% RSLogix 500 project ANALOG PID HEATER CONTROL.RSS, saved by version 8.30.00.16 %
PROJECT "HEATER"    % processor: Bul.1763 MicroLogix 1100 Series B %

PROGRAM FILES
  LAD 2   6 rungs

DATA FILES
  O0 OUTPUT  8 elements
  I1 INPUT  15 elements
  S2 STATUS  66 elements
  B3 BINARY  1 elements
  T4 TIMER  1 elements
  C5 COUNTER  1 elements
  R6 CONTROL  1 elements
  N7 INTEGER  2 elements
  F8 FLOAT  1 elements
  PD9   1 elements

LADDER 2
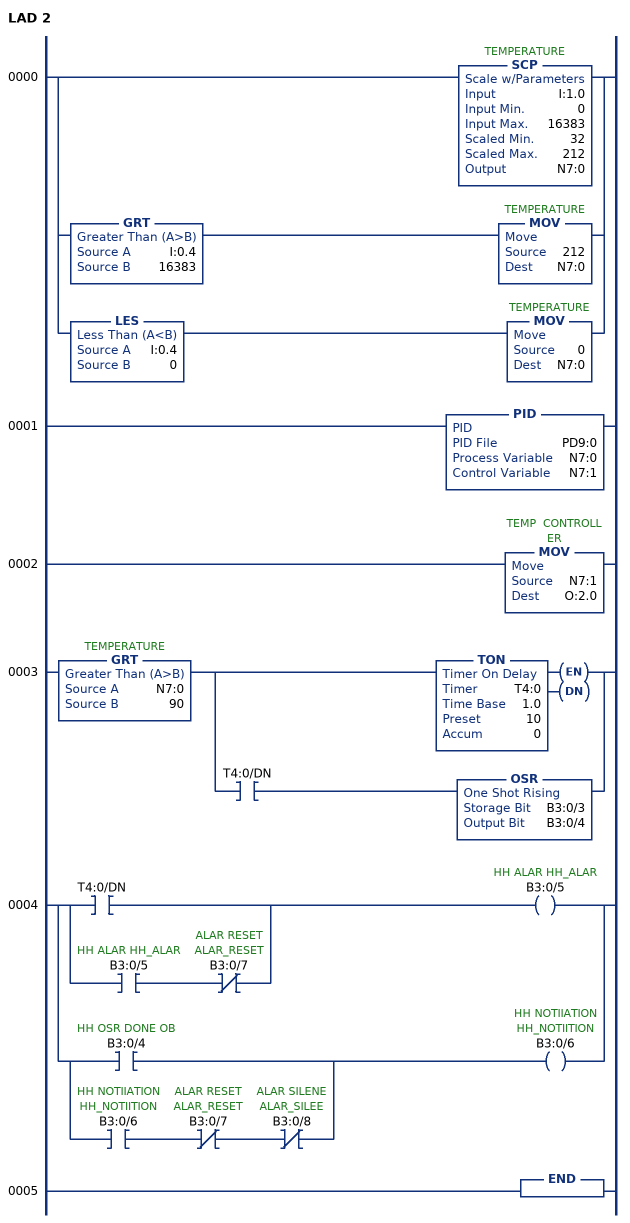
% Rung: 0 %
SOR BST SCP I:1.0 0 16383 32 212 N7:0 NXB GRT I:0.4 16383 MOV 212 N7:0 NXB LES I:0.4 0 MOV 0 N7:0 BND EOR
%   N7:0  "TEMPERATURE" %
% Rung: 1 %
SOR PID PD9:0 N7:0 N7:1 EOR
%   N7:0  "TEMPERATURE" %
% Rung: 2 %
SOR MOV N7:1 O:2.0 EOR
%   O:2.0  "TEMP  CONTROLLER" %
% Rung: 3 %
SOR GRT N7:0 90 BST TON T4:0 1.0 10 0 NXB XIC T4:0/DN OSR B3:0/3 B3:0/4 BND EOR
%   N7:0  "TEMPERATURE" %
%   B3:0/4  "HH OSR DONE OB" %
% Rung: 4 %
SOR BST BST XIC T4:0/DN NXB XIC B3:0/5 XIO B3:0/7 BND OTE B3:0/5 NXB BST XIC B3:0/4 NXB XIC B3:0/6 XIO B3:0/7 XIO B3:0/8 BND OTE B3:0/6 BND EOR
%   B3:0/5  HH_ALAR  "HH ALAR" %
%   B3:0/7  ALAR_RESET  "ALAR RESET" %
%   B3:0/4  "HH OSR DONE OB" %
%   B3:0/6  HH_NOTIITION  "HH NOTIIATION" %
%   B3:0/8  ALAR_SILEE  "ALAR SILENE" %
% Rung: 5 %
SOR END EOR

DATA TABLE (non-zero values as saved)
DATA T4
% .PRE .ACC %
% T4:0 % 10 0
DATA N7
% N7:0 % 32 0
